{attribute 'GeneratedUsingTerminal: EK1122-0000-0018'}
{attribute addProperty BoxType "EK1122-0000-0018"}
{attribute addProperty Id "Beckhoff_ELM36xxsub_EK1100EK1100_1FC0878B2"}
{attribute addProperty CRC "2444466482"}
{attribute addProperty Size "2"}
TYPE Beckhoff_ELM36xxEK1122_91B39932 EXTENDS EK1122_1FC0878B :
STRUCT
	{attribute addProperty Name "Beckhoff_ELM36xxsub_EK1100"}
	Beckhoff_ELM36xxsub_EK1100 : EK1100_1FC0878B;
END_STRUCT
END_TYPE

(* stored: Version 1.2.0.0, ProductVersion 3.1.4024.9
   DUT Beckhoff_ELM36xxEK1122_91B39932: Id {7954b5a2-821b-4574-bbbd-3f23891725e0} *)
